// TIA Portal V20 export
FUNCTION "LER_TwoWayActuaorCommand" : Void   // FC86, LAD
// stored: Access Published, SetENOAutomatically false
   VAR_INPUT
      enable : Bool;
   END_VAR
   VAR_IN_OUT
      Command : USInt;
      TwoWayActuator : "LBC_typeTwoWayActuatorControlNode";
   END_VAR
   VAR CONSTANT
      CommandReset : USInt;
      CommandHomePos : USInt := 1;
      CommandWorkPos : USInt := 2;
   END_VAR
BEGIN

REGION Network 1: Rising edge: Move actuator to home position
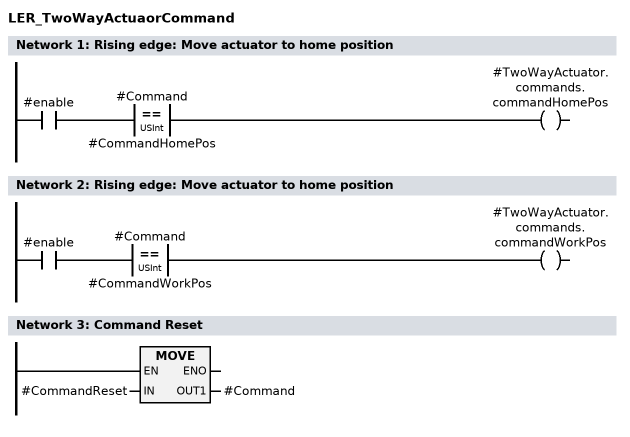
   RUNG wire#powerrail
      Contact( #enable )
      { S7_Templates := "SrcType := USInt" } EQ_Contact(in1 := #Command, in2 := #CommandHomePos)
      Coil( #TwoWayActuator.commands.commandHomePos )
   END_RUNG
   // the same network as SCL:
   #TwoWayActuator.commands.commandHomePos := #enable AND (#Command = #CommandHomePos);
END_REGION

REGION Network 2: Rising edge: Move actuator to home position
   RUNG wire#powerrail
      Contact( #enable )
      { S7_Templates := "SrcType := USInt" } EQ_Contact(in1 := #Command, in2 := #CommandWorkPos)
      Coil( #TwoWayActuator.commands.commandWorkPos )
   END_RUNG
   // the same network as SCL:
   #TwoWayActuator.commands.commandWorkPos := #enable AND (#Command = #CommandWorkPos);
END_REGION

REGION Network 3: Command Reset
   RUNG wire#powerrail
      Move(in := #CommandReset, out1 => #Command)
   END_RUNG
   // the same network as SCL:
   #Command := #CommandReset;
END_REGION
END_FUNCTION
